{attribute 'linkalways'} 
{attribute 'no_explicit_call' := 'This FB is a CLASS and must be accessed using methods or properties'}
{attribute 'enable_dynamic_creation'}
FUNCTION_BLOCK _UDINT EXTENDS NumericDatatypeBase
VAR
	localData : UDINT;
	activeData : REFERENCE TO UDINT REF= localData;
END_VAR

PROPERTY PUBLIC Address : PVOID
GET
Address := ADR(activeData);
END_GET
END_PROPERTY

METHOD PUBLIC ClearReference
VAR_INPUT
END_VAR
activeData REF= localData;
END_METHOD

METHOD PUBLIC Clone : I_Datatype
VAR
    pClone : POINTER TO _UDINT;
END_VAR
pClone := __NEW(_UDINT(InitialValue := Value));
Clone := pClone^;
END_METHOD

METHOD FB_init : BOOL
VAR_INPUT
	bInitRetains : BOOL; // if TRUE, the retain variables are initialized (warm start / cold start)
	bInCopyCode : BOOL;  // if TRUE, the instance afterwards gets moved into the copy code (online change)
	InitialValue : UDINT;
END_VAR
localData := InitialValue;
END_METHOD

PROPERTY PUBLIC IsFloat : BOOL
GET
IsFloat := FALSE;
END_GET
END_PROPERTY

PROPERTY PUBLIC IsSigned : BOOL
GET
IsSigned := FALSE;
END_GET
END_PROPERTY

METHOD PUBLIC MakeReferenceTo
VAR_INPUT
	ReferenceTarget : REFERENCE TO UDINT;
END_VAR
activeData REF= ReferenceTarget;
END_METHOD

PROPERTY PUBLIC MaxValue : UDINT
GET
MaxValue :=  DatatypeLimits.UDINT_MAX_VALUE;
END_GET
END_PROPERTY

PROPERTY PUBLIC MinValue : UDINT
GET
MinValue := DatatypeLimits.UDINT_MIN_VALUE;
END_GET
END_PROPERTY

METHOD PROTECTED SerializeMaxValue
VAR_INPUT
	Serializer : I_Serializer;
END_VAR
Serializer.AddUdint(MaxValue);
END_METHOD

METHOD PROTECTED SerializeMinValue
VAR_INPUT
	Serializer : I_Serializer;
END_VAR
Serializer.AddUdint(MinValue);
END_METHOD

METHOD PUBLIC SerializeWith
VAR_INPUT
	Serializer : I_Serializer;
END_VAR
Serializer.AddUdint(activeData);
END_METHOD

PROPERTY PUBLIC Size : UDINT
GET
Size := SIZEOF(activeData);
END_GET
END_PROPERTY

METHOD TryDeserializeFrom : BOOL
VAR_INPUT
	Deserializer : I_Deserializer;
	Feedback : I_DeserializerFeedback;
END_VAR
TryDeserializeFrom := Deserializer.TryGetUdint(activeData, Feedback);
END_METHOD

METHOD TryMakeReferenceTo : BOOL
VAR_INPUT
	Target : I_Datatype;
END_VAR
VAR
	pTargetData : POINTER TO UDINT;
END_VAR
IF NOT (Target.TypeName = TypeName) THEN
	RETURN;
END_IF

pTargetData := Target.Address;
activeData REF= pTargetData^;
TryMakeReferenceTo := TRUE;
END_METHOD

PROPERTY PUBLIC TypeName : T_MAXSTRING
GET
TypeName := 'UDINT';
END_GET
END_PROPERTY

PROPERTY PUBLIC Value : REFERENCE TO UDINT
GET
Value REF= activeData;
END_GET
END_PROPERTY

END_FUNCTION_BLOCK

(* stored: Version 1.1.0.1, ProductVersion 3.1.4024.12
   POU _UDINT: Id {33df45f2-c623-4e8f-9a45-837fa33bdb08}, SpecialFunc None
   Folder Constructor: Id {fa10fb2a-0e3b-4eb4-b0fd-4bac30e4b7ef}
   Folder Protected: Id {30ac8c27-c61c-4404-819e-0090d4d9f95f}
   Property Address: Id {29238022-4923-4acb-9df0-cd263a10ad16}
   Get Get: Id {73736b5c-f03a-45d5-9d03-9f39c42f2bcc}
   Method ClearReference: Id {573c11cc-055f-4ab4-8809-b95724d5c50c}
   Method Clone: Id {0d48dc1b-d691-48ec-8323-a05e219f634e}
   Method FB_init: Id {5043c549-e026-44ca-8fff-68547159acc6}
   Property IsFloat: Id {c214fc70-d07a-42c2-9bb0-4321605b2f93}
   Get Get: Id {7801af26-a89e-4373-9647-bef3f9e17a41}
   Property IsSigned: Id {2aebf7e8-f67a-4cd8-b40b-eea14729f1fc}
   Get Get: Id {655b7264-4181-4b56-ace7-fa519768c185}
   Method MakeReferenceTo: Id {3ec1b088-8843-45a5-a20f-507c2a25fc11}
   Property MaxValue: Id {f7f661b8-45f8-42e4-a23a-6b88308d6e05}
   Get Get: Id {d61aa2c4-4dbe-4423-9840-2d1676675210}
   Property MinValue: Id {28e4e9ec-c6ce-422e-b78d-ff22b8b39b17}
   Get Get: Id {117cae1b-e957-4156-bcf8-a7a74ce3c4eb}
   Method SerializeMaxValue: Id {c3bf67fb-5699-4bbf-94ac-00981b7d7cbd}
   Method SerializeMinValue: Id {366bfebe-abd0-487b-99aa-a58b968135dd}
   Method SerializeWith: Id {89c10341-24db-4e48-aa66-9cfdd3e854ae}
   Property Size: Id {abb72fd2-ade6-4d5c-acc9-20396d77423a}
   Get Get: Id {ba7ff353-ba1b-4e59-9eb2-14b42ddab42b}
   Method TryDeserializeFrom: Id {558846e9-23ed-42bd-a566-ea76a84f6c46}
   Method TryMakeReferenceTo: Id {3b69d30b-e89e-4a22-b3e9-c80605793d1c}
   Property TypeName: Id {72092dae-bca7-43a1-82b2-205025bcb5cd}
   Get Get: Id {84fb3bb5-24cc-48f7-8fd6-5d7678ac61bb}
   Property Value: Id {f9e1bfb5-db30-4dce-a5bc-8eb3e24090ae}
   Get Get: Id {592b7321-5776-4624-a68f-5a851ff2b2ff} *)
